// TwinCAT 3 PLC project PLC3
// ProgramVersion: 3.1.4022.3
// libraries:
//   Tc2_Standard, * (Beckhoff Automation GmbH)
//   Tc2_System, * (Beckhoff Automation GmbH)
//   Tc3_Module, * (Beckhoff Automation GmbH)
// project tree:
//   DUTs/ DeviceState.TcDUT
//   GVLs/ GVL_IO.TcGVL
//   / PlcTask.TcTTO
//   POUs/ MAIN.TcPOU
// real-time tasks:
//   TASK PlcTask: cycle T#10ms, priority 20, ADS port 350
// I/O:
//   DEVICE Device 3 (EtherCAT), AmsNetId 145.85.88.31.4.1
//     Term 7 (EK1100) [EK1100 EtherCAT Coupler (2A E-Bus)]
//       Term 8 (EL1809) [EL1809 16Ch. Dig. Input 24V, 3ms]
//       Term 9 (EL1809) [EL1809 16Ch. Dig. Input 24V, 3ms]
//       Term 10 (EL2809) [EL2809 16Ch. Dig. Output 24V, 0.5A]
//       Term 11 (EL2809) [EL2809 16Ch. Dig. Output 24V, 0.5A]
//       Term 6 (EL9011) [EL9011 End Terminal]
// variable links:
//   PLC3/PLC3 Instance <-> Device 3 (EtherCAT)/Term 7 (EK1100)/Term 10 (EL2809)
//     PlcTask Outputs/GVL_IO.Aplus_Vert_axis_downwards <-> Channel 2/Output
//     PlcTask Outputs/GVL_IO.BR_Alarm_light <-> Channel 1/Output
//     PlcTask Outputs/GVL_IO.DRIVEX_MOVE_tableX <-> Channel 10/Output
//     PlcTask Outputs/GVL_IO.DRIVEY_MOVE_translY <-> Channel 16/Output
//     PlcTask Outputs/GVL_IO.HOLD_STOP_tableX_AND_translY <-> Channel 9/Output
//     PlcTask Outputs/GVL_IO.INX0_from_Input0_tableX <-> Channel 4/Output
//     PlcTask Outputs/GVL_IO.INX1_from_Input1_tableX <-> Channel 5/Output
//     PlcTask Outputs/GVL_IO.INX2_from_Input2_tableX <-> Channel 6/Output
//     PlcTask Outputs/GVL_IO.INY0_from_Input0_translY <-> Channel 11/Output
//     PlcTask Outputs/GVL_IO.INY1_from_Input1_translY <-> Channel 12/Output
//     PlcTask Outputs/GVL_IO.INY2_from_Input2_translY <-> Channel 13/Output
//     PlcTask Outputs/GVL_IO.SETUPX_ORIGIN_tableX <-> Channel 8/Output
//     PlcTask Outputs/GVL_IO.SETUPY_ORIGIN_translY <-> Channel 15/Output
//     PlcTask Outputs/GVL_IO.SVONX_SERVO_ON_tableX <-> Channel 7/Output
//     PlcTask Outputs/GVL_IO.SVONY_SERVO_ON_translY <-> Channel 14/Output
//     PlcTask Outputs/GVL_IO.Vplus_Vacuum_start <-> Channel 3/Output
//   PLC3/PLC3 Instance <-> Device 3 (EtherCAT)/Term 7 (EK1100)/Term 8 (EL1809)
//     PlcTask Inputs/GVL_IO.ALARMX_ALARM_tableX <-> Channel 11/Input
//     PlcTask Inputs/GVL_IO.ALARMY_ALARM_translationY <-> Channel 15/Input
//     PlcTask Inputs/GVL_IO.Auto_I_Manual_II_switch <-> Channel 3/Input
//     PlcTask Inputs/GVL_IO.BUSYX_BUSY_tableX <-> Channel 9/Input
//     PlcTask Inputs/GVL_IO.BUSYY_BUSY_traslationY <-> Channel 13/Input
//     PlcTask Inputs/GVL_IO.EMERX_EMERGENCY_tableX <-> Channel 12/Input
//     PlcTask Inputs/GVL_IO.EMERY_EMERGENCY_translationY <-> Channel 16/Input
//     PlcTask Inputs/GVL_IO.Reset_button <-> Channel 4/Input
//     PlcTask Inputs/GVL_IO.SETONX_ORIGIN_tableX <-> Channel 10/Input
//     PlcTask Inputs/GVL_IO.SETONY_ORIGIN_translationY <-> Channel 14/Input
//     PlcTask Inputs/GVL_IO.Start_button <-> Channel 1/Input
//     PlcTask Inputs/GVL_IO.Stop_button <-> Channel 2/Input
//     PlcTask Inputs/GVL_IO.a_0_Vertical_Zaxis_upward <-> Channel 5/Input
//     PlcTask Inputs/GVL_IO.a_1_Vertical_Zaxis_downward <-> Channel 6/Input
//     PlcTask Inputs/GVL_IO.dp1_Can_detection <-> Channel 7/Input
//     PlcTask Inputs/GVL_IO.dp2_Cover_detection <-> Channel 8/Input

CONFIGURATION PLC3
    RESOURCE PLC ON TwinCAT3
        TASK PlcTask(INTERVAL := T#10ms, PRIORITY := 20);
        PROGRAM MAIN WITH PlcTask : MAIN;
    END_RESOURCE
END_CONFIGURATION

// ---- DUTs/DeviceState.TcDUT
{attribute 'qualified_only'}
{attribute 'strict'}
TYPE DeviceState :
(
	Init := 0,
	Idle := 1,
	MoveToPickUp := 2,
	PickUpDown := 3,
	PickUpUp := 4,
	MoveX := 5,
	MoveY := 6,
	DropDown := 7,
	DropUp := 8,
	PalletFull := 9
);
END_TYPE

// ---- GVLs/GVL_IO.TcGVL
{attribute 'qualified_only'}     // Do not remove this line
VAR_GLOBAL
// Input module EL1809	
    Start_button                 AT %I* :BOOL;
    Stop_button                  AT %I* :BOOL;
    Auto_I_Manual_II_switch      AT %I* :BOOL;
    Reset_button                 AT %I* :BOOL;
    a_0_Vertical_Zaxis_upward    AT %I* :BOOL;
    a_1_Vertical_Zaxis_downward  AT %I* :BOOL;
    dp1_Can_detection            AT %I* :BOOL;
    dp2_Cover_detection          AT %I* :BOOL;
    BUSYX_BUSY_tableX            AT %I* :BOOL;
    SETONX_ORIGIN_tableX         AT %I* :BOOL;
    ALARMX_ALARM_tableX          AT %I* :BOOL;
    EMERX_EMERGENCY_tableX       AT %I* :BOOL;
    BUSYY_BUSY_traslationY       AT %I* :BOOL;
    SETONY_ORIGIN_translationY   AT %I* :BOOL;
    ALARMY_ALARM_translationY    AT %I* :BOOL;
    EMERY_EMERGENCY_translationY AT %I* :BOOL;
//========================================
	INPUTchannel_01_SPARE        AT %I* :BOOL;
	INPUTchannel_02_SPARE        AT %I* :BOOL;
	INPUTchannel_03_SPARE        AT %I* :BOOL;
	INPUTchannel_04_SPARE        AT %I* :BOOL;
	INPUTchannel_05_SPARE        AT %I* :BOOL;
	INPUTchannel_06_SPARE        AT %I* :BOOL;
	INPUTchannel_07_SPARE        AT %I* :BOOL;
	INPUTchannel_08_SPARE        AT %I* :BOOL;
	INPUTchannel_09_SPARE        AT %I* :BOOL;
	INPUTchannel_10_SPARE        AT %I* :BOOL;
	INPUTchannel_11_SPARE        AT %I* :BOOL;
	INPUTchannel_12_SPARE        AT %I* :BOOL;
	INPUTchannel_13_SPARE        AT %I* :BOOL;
	INPUTchannel_14_SPARE        AT %I* :BOOL;
	INPUTchannel_15_SPARE        AT %I* :BOOL;
	INPUTchannel_16_SPARE        AT %I* :BOOL;
//========================================
	BR_Alarm_light               AT %Q* :BOOL;
    Aplus_Vert_axis_downwards    AT %Q* :BOOL;
    Vplus_Vacuum_start           AT %Q* :BOOL;
    INX0_from_Input0_tableX      AT %Q* :BOOL;
    INX1_from_Input1_tableX      AT %Q* :BOOL;
    INX2_from_Input2_tableX      AT %Q* :BOOL;
    SVONX_SERVO_ON_tableX        AT %Q* :BOOL;
    SETUPX_ORIGIN_tableX         AT %Q* :BOOL;
    HOLD_STOP_tableX_AND_translY AT %Q* :BOOL;
    DRIVEX_MOVE_tableX           AT %Q* :BOOL;
    INY0_from_Input0_translY     AT %Q* :BOOL;
    INY1_from_Input1_translY     AT %Q* :BOOL;
    INY2_from_Input2_translY     AT %Q* :BOOL;
    SVONY_SERVO_ON_translY       AT %Q* :BOOL;
    SETUPY_ORIGIN_translY        AT %Q* :BOOL;
    DRIVEY_MOVE_translY          AT %Q* :BOOL;
//============================================
    OUTPUTchannel_01_SPARE       AT %Q* :BOOL;
    OUTPUTchannel_02_SPARE       AT %Q* :BOOL;
    OUTPUTchannel_03_SPARE       AT %Q* :BOOL;
    OUTPUTchannel_04_SPARE       AT %Q* :BOOL;
    OUTPUTchannel_05_SPARE       AT %Q* :BOOL;
    OUTPUTchannel_06_SPARE       AT %Q* :BOOL;
    OUTPUTchannel_07_SPARE       AT %Q* :BOOL;
    OUTPUTchannel_08_SPARE       AT %Q* :BOOL;
    OUTPUTchannel_00_SPARE       AT %Q* :BOOL;
    OUTPUTchannel_10_SPARE       AT %Q* :BOOL;
    OUTPUTchannel_11_SPARE       AT %Q* :BOOL;
    OUTPUTchannel_12_SPARE       AT %Q* :BOOL;
    OUTPUTchannel_13_SPARE       AT %Q* :BOOL;
    OUTPUTchannel_14_SPARE       AT %Q* :BOOL;
    OUTPUTchannel_15_SPARE       AT %Q* :BOOL;
    OUTPUTchannel_16_SPARE       AT %Q* :BOOL;
END_VAR

// ---- POUs/MAIN.TcPOU
PROGRAM MAIN
VAR
	Timer1 :TON;
	Timer2 :TON;
	Start  :BOOL;
	Full   :BOOL;
	PosX   :INT;
	PosY   :INT;
	CurrentState  :DeviceState;
END_VAR

CASE CurrentState OF
	DeviceState.Init:
		GVL_IO.SVONX_SERVO_ON_tableX 	  := TRUE;
		GVL_IO.SVONY_SERVO_ON_translY 	  := TRUE;
		GVL_IO.SETONX_ORIGIN_tableX 	  := TRUE;
		GVL_IO.SETONY_ORIGIN_translationY := TRUE;
		
		Timer1(IN:= TRUE, PT:= T#60MS);
		//TO IDLE
		IF Timer1.Q AND NOT GVL_IO.BUSYX_BUSY_tableX AND NOT GVL_IO.BUSYY_BUSY_traslationY AND GVL_IO.SETONX_ORIGIN_tableX AND GVL_IO.SETONY_ORIGIN_translationY THEN
			CurrentState := DeviceState.Idle;
			END_IF	
			
	DeviceState.Idle:
		//TO MOVE TO PICK UP
		IF FULL THEN
			CurrentState := DeviceState.PalletFull;
			END_IF
		//TO IDLE
		IF NOT GVL_IO.dp2_Cover_detection THEN // AND MSG.Received AND MSG.Send(NoCover) !!!!!!!!!!!!!!!!!!!!!!!!!!!!!!!!!!!!
			CurrentState := DeviceState.Idle;
			END_IF
		//TO PALLET FULL
		IF GVL_IO.dp1_Can_detection AND GVL_IO.dp2_Cover_detection AND NOT Full THEN // AND MSG.Received !!!!!!!!!!!!!!!!!!!!
			CurrentState := DeviceState.PalletFull;
			END_IF
		
	DeviceState.MoveToPickUp:
		GVL_IO.INY0_from_Input0_translY := TRUE;
		GVL_IO.INY1_from_Input1_translY := FALSE;	
		GVL_IO.INY2_from_Input2_translY := TRUE;
		
		GVL_IO.INX0_from_Input0_tableX := FALSE;
		GVL_IO.INX1_from_Input1_tableX := FALSE;	
		GVL_IO.INX2_from_Input2_tableX := TRUE;
		
		Timer1(IN:= TRUE, PT:= T#15MS);
		IF Timer1.Q THEN
			GVL_IO.DRIVEY_MOVE_translY := TRUE;
			GVL_IO.DRIVEX_MOVE_tableX  := TRUE;
			Timer2(IN:= TRUE, PT:= T#150MS);
 			END_IF
		//TO PICK-UP DOWN
		IF Timer2.Q AND NOT GVL_IO.BUSYY_BUSY_traslationY AND NOT GVL_IO.BUSYX_BUSY_tableX THEN
			CurrentState := DeviceState.PickUpDown;
			END_IF
	
	DeviceState.PickUpDown:
		IF GVL_IO.a_0_Vertical_Zaxis_upward THEN
			GVL_IO.Aplus_Vert_axis_downwards := TRUE;
			END_IF
		IF GVL_IO.a_1_Vertical_Zaxis_downward THEN
			GVL_IO.Vplus_Vacuum_start := TRUE;
			Timer1(IN:= TRUE, PT:= T#10MS);
			END_IF
		//TO PICK-UP UP
		IF Timer1.Q THEN
			CurrentState := DeviceState.PickUpUp;
			END_IF
	
	DeviceState.PickUpUp:
		GVL_IO.Aplus_Vert_axis_downwards := FALSE;
		//TO MOVE X
		IF GVL_IO.a_0_Vertical_Zaxis_upward THEN
			CurrentState := DeviceState.MoveX;
			END_IF		
	
	DeviceState.MoveX:
		//SwitchMoveX(); !!!!!!!!!!!!!!!!!!!!!!!!!!!!!!!!!!!!!!!!!!!!!!!!!!!!!!!!!!!!!!!!!!!!!!!!!!!!!!!!!!!!!!!!!!!
		
		PosX := PosX + 1;
		IF PosX >= 4 THEN
			PosX := 0; 
			PosY := PosY + 1;
			END_IF	
		IF PosY >= 4 AND PosX >= 4 THEN
		 	Full := TRUE;
			END_IF	
		//TO MOVE Y
		IF NOT GVL_IO.BUSYX_BUSY_tableX THEN
			CurrentState := DeviceState.MoveY;
			END_IF
	
	DeviceState.MoveY:
		//SwitchMoveY(); !!!!!!!!!!!!!!!!!!!!!!!!!!!!!!!!!!!!!!!!!!!!!!!!!!!!!!!!!!!!!!!!!!!!!!!!!!!!!!!!!!!!!!!!!!
		
		//TO DROP DOWN
		IF NOT GVL_IO.BUSYY_BUSY_traslationY THEN
			CurrentState := DeviceState.DropDown;
			END_IF
			
	DeviceState.DropDown:
		IF GVL_IO.a_0_Vertical_Zaxis_upward THEN
			GVL_IO.Aplus_Vert_axis_downwards := TRUE;
			END_IF
		IF GVL_IO.a_1_Vertical_Zaxis_downward THEN
			GVL_IO.Vplus_Vacuum_start := TRUE;
			Timer1(IN:= TRUE, PT:= T#10MS);
			END_IF
		//TO DROP UP
		IF NOT Timer1.Q THEN
			CurrentState := DeviceState.DropUp;
			END_IF
	
	DeviceState.DropUp:
		IF GVL_IO.a_1_Vertical_Zaxis_downward THEN
			GVL_IO.Aplus_Vert_axis_downwards := FALSE;
			END_IF
		//TO IDLE
		IF GVL_IO.a_0_Vertical_Zaxis_upward THEN
			CurrentState := DeviceState.Idle;
			END_IF
	
	DeviceState.PalletFull:
		//SendMSG(FULL); !!!!!!!!!!!!!!!!!!!!!!!!!!!!!!!!!!!!!!!!!!!!!!!!!
		GVL_IO.BR_Alarm_light := TRUE;
END_CASE

END_PROGRAM
